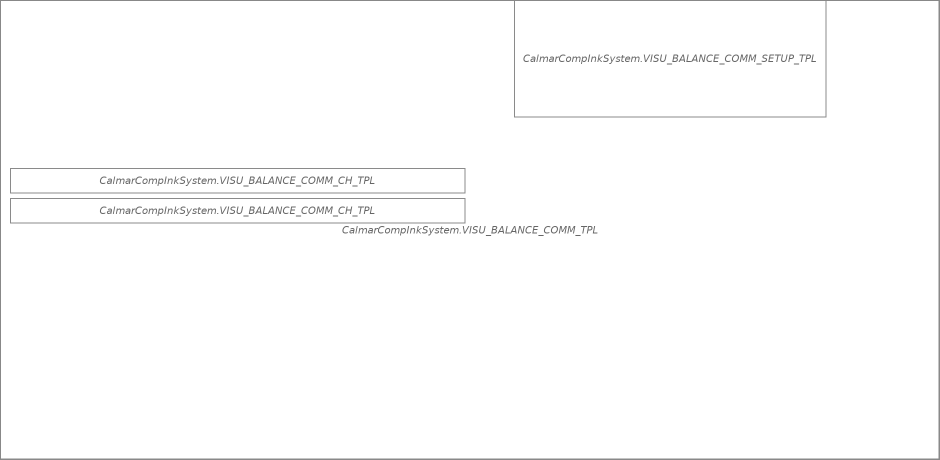
VISUALIZATION VISU_COMM_BALANCE  // 940x460
    Frame (0,0 940x460)
        shows CalmarCompInkSystem.VISU_BALANCE_COMM_TPL(m_ModId_FbBalanceComm := PRG_INK.FB_BalanceLink)
    Frame (514,0 312x117)
        shows CalmarCompInkSystem.VISU_BALANCE_COMM_SETUP_TPL(m_ModId_FbBalanceComm := PRG_INK.FB_BalanceLink)
    Frame (10,168 455x25)
        shows CalmarCompInkSystem.VISU_BALANCE_COMM_CH_TPL(m_Idx := 1, m_ModId_StAdsStorageTank := PRG_INK.sAdsIkInkStorageTank[1], m_ModId_StInkDefinition := PRG_INK.sL_InkTable[1], m_ModId_FbBalanceComm := PRG_INK.FB_BalanceLink)
    Frame (10,198 455x25)
        shows CalmarCompInkSystem.VISU_BALANCE_COMM_CH_TPL(m_Idx := 2, m_ModId_StAdsStorageTank := PRG_INK.sAdsIkInkStorageTank[2], m_ModId_StInkDefinition := PRG_INK.sL_InkTable[2], m_ModId_FbBalanceComm := PRG_INK.FB_BalanceLink)
END_VISUALIZATION

(* stored: Version 1.1.0.1, ProductVersion 3.1.4024.9
   Visu VISU_COMM_BALANCE: Id {1b036466-4acd-4626-93cf-2c7394fb09a3} *)
